PROGRAM MAIN

ResetWriteData(AdsNet6.WriteTestData.WriteGenericUpdatesTheValueInPlc);
ResetWriteData(AdsNet6.WriteTestData.WriteGenericUpdatesTheValueInPlcAsync);
ResetWriteData(AdsNet6.WriteTestData.WriteMultipleUpdatesTheValueInPlc);
ResetWriteData(AdsNet6.WriteTestData.WriteMultipleUpdatesTheValueInPlcAsync);
ResetWriteData(AdsNet6.WriteTestData.WriteUpdatesTheValueInPlc);
ResetWriteData(AdsNet6.WriteTestData.WriteUpdatesTheValueInPlcAsync);

ResetWriteData(AdsNet7.WriteTestData.WriteGenericUpdatesTheValueInPlc);
ResetWriteData(AdsNet7.WriteTestData.WriteGenericUpdatesTheValueInPlcAsync);
ResetWriteData(AdsNet7.WriteTestData.WriteMultipleUpdatesTheValueInPlc);
ResetWriteData(AdsNet7.WriteTestData.WriteMultipleUpdatesTheValueInPlcAsync);
ResetWriteData(AdsNet7.WriteTestData.WriteUpdatesTheValueInPlc);
ResetWriteData(AdsNet7.WriteTestData.WriteUpdatesTheValueInPlcAsync);

ResetWriteData(OpcNet6.WriteTestData.WriteGenericUpdatesTheValueInPlc);
ResetWriteData(OpcNet6.WriteTestData.WriteGenericUpdatesTheValueInPlcAsync);
ResetWriteData(OpcNet6.WriteTestData.WriteMultipleUpdatesTheValueInPlc);
ResetWriteData(OpcNet6.WriteTestData.WriteMultipleUpdatesTheValueInPlcAsync);
ResetWriteData(OpcNet6.WriteTestData.WriteUpdatesTheValueInPlc);
ResetWriteData(OpcNet6.WriteTestData.WriteUpdatesTheValueInPlcAsync);

ResetWriteData(OpcNet7.WriteTestData.WriteGenericUpdatesTheValueInPlc);
ResetWriteData(OpcNet7.WriteTestData.WriteGenericUpdatesTheValueInPlcAsync);
ResetWriteData(OpcNet7.WriteTestData.WriteMultipleUpdatesTheValueInPlc);
ResetWriteData(OpcNet7.WriteTestData.WriteMultipleUpdatesTheValueInPlcAsync);
ResetWriteData(OpcNet7.WriteTestData.WriteUpdatesTheValueInPlc);
ResetWriteData(OpcNet7.WriteTestData.WriteUpdatesTheValueInPlcAsync);

END_PROGRAM

(* stored: Version 1.1.0.1, ProductVersion 3.1.4024.12
   POU MAIN: Id {65800fe3-bb5f-43d1-b26a-4a3b6ac53c7a}, SpecialFunc None *)
